(* IEC 61131-3 sources: test/SharedPlc, 5 files *)

(* ---- LPHD_Time.gvl ---- *)
VAR_GLOBAL
	DtTmAct 			: DT; 		(* --- Actual local time without summer time shift *)
	DtTmActSec 			: DINT;		(* --- Actual local time in second since 1.1.1970 *)
	DtTmActUtc 			: DT; 		(* --- Actual UTC Date and Time from the control system *)
	DtTmActUtcSec 		: DINT; 	(* --- Actual UTC Date and Time from the control system in seconds since 1.1.1970 *)
	DtTmShStri			: STRING;	(* --- Timezone shift from UTC in the format 'GMT+00:00'*)
	DtTmShSec			: DINT;		(* --- Timezone shift in seconds *)
	DtTmShM				: DINT;		(* --- Timezone shift in minutes *)
END_VAR

(* ---- SwitchIO.st ---- *)
FUNCTION SwitchIO : BOOL
VAR_INPUT
                Val:        BOOL;
                Switch: DINT;
END_VAR

VAR

END_VAR

CASE Switch OF
                -1: SwitchIO := Val XOR TRUE;
                0:  SwitchIO := FALSE;
                1:  SwitchIO := TRUE;
                2:  SwitchIO := Val;
END_CASE

END_FUNCTION

(* ---- TonSec.st ---- *)
FUNCTION_BLOCK TonSec
VAR_INPUT
	In		: BOOL;
	PTs		: DWORD; (* --- Time in seconds *)
END_VAR
VAR_OUTPUT
	ETs	:	DWORD;
	Q		: BOOL;
	PTDT	: DT;
	ETDT	: DT;	(* --- Time in seconds *)
END_VAR
VAR
	Str		: R_TRIG;
	StrTm 	: DT;
END_VAR

Str(S1 := In);
IF Str.Q0 THEN
	StrTm := DtTmActUtc;
END_IF

PTDT := UDINT_TO_DT(DT_TO_UDINT(StrTm) + PTs);
IF In THEN
	IF ETDT < PTDT   THEN

		ETDT := DtTmActUtc;
		ETs := PTs - (DT_TO_UDINT(PTDT) - DT_TO_UDINT(ETDT));
	END_IF

	IF ETDT >= PTDT THEN
		Q := TRUE;
	END_IF
ELSE
	ETs		:=	0;
	ETDT	:=	BYTE_TO_DT(0);
	Q		:=	FALSE;
END_IF

END_FUNCTION_BLOCK

(* ---- UpDnCnt.st ---- *)
FUNCTION_BLOCK UpDnCnt

VAR_INPUT
	IN		: BOOL;
	Cyc		: UDINT;
	RsCond	: INT;
END_VAR
VAR_OUTPUT
	OUT		: BOOL;
	CntEnd	: BOOL;
END_VAR
VAR
	Cnt: UDINT;
END_VAR

(* --- Reset Condition 0: Out will be FALSE, if IN FALSE *)
(* --- Reset Condition 1: Out will be FALSE, if IN FALSE and the time was counted down *)

IF (IN) THEN
	IF (Cnt >= Cyc) THEN
		Cnt := Cyc;
		OUT := TRUE;
	ELSE
		Cnt := Cnt + 1;
	END_IF
ELSE
	IF (Cnt <= 0) THEN
		Cnt := 0;
		OUT := FALSE;
	ELSE
		Cnt := Cnt - 1;
	END_IF

	IF(RsCond = 0)THEN
		OUT := FALSE;
	END_IF
END_IF

CntEnd := Cnt >= Cyc;

END_FUNCTION_BLOCK

(* ---- TimeHdl.st ---- *)
PROGRAM TimeHdl
VAR
	timespec_microseconds_Ds	: timespec_microseconds;
	DtOld						: DT;
	DtTmActLoc					: DT;
	SysTmUsec					: UDINT;
	USecOld						: UDINT;
	USecAct						:UDINT;
END_VAR
VAR_OUTPUT
	DTMS : DTMS;
END_VAR

(* --- Get time from system *)
clock_gettime(ADR(timespec_microseconds_Ds),TIMESPEC_RESOLUTION_MICROSECONDS,CLOCK_ID_CLOCK_RTCNANO);

DtTmActLoc := timespec_microseconds_Ds.dateAndTime;

(* WppTimeShiftMinutes_GDi: Wird aus der Monitoring Vorgabe in TimeZone_GpSt geholt *)
DTMS.DateAndTime := DINT_TO_DT(DT_TO_DINT(DtTmActLoc) + DtTmShSec);

(* --- SysTmUsec are in s from CPU start *)
SysTmUsec			:= timespec_microseconds_Ds.microseconds;
USecAct  			:= ((USecAct + ABS(SysTmUsec - USecOld)) MOD 1000000);
DTMS.Millisecond 	:= UDINT_TO_UINT(USecAct / 1000);

IF (TIME_TO_BOOL (ABS(DTMS.DateAndTime - DtOld))) THEN
	USecAct := 0;
END_IF

USecOld := SysTmUsec;
DtOld := DTMS.DateAndTime;

DtTmAct 		:= DTMS.DateAndTime;				(* --- Actual local time without summer time shift *)
DtTmActSec 		:= DT_TO_UDINT(DtTmAct);			(* --- Actual local time in second since 1.1.1970 *)
DtTmActUtc 		:= Tcs_RTC_GetDateAndTime(0);		(* --- Actual UTC Date and Time from the control system *)
DtTmActUtcSec 	:= DT_TO_UDINT(DtTmActUtc);			(* --- Actual UTC Date and Time from the control system in seconds since 1.1.1970 *)

(* TODO: check where we can get this information*)
(*ActDateAndTimeDST_GDt 	:=*) 						(* --- Actual local time with summer time shift *)

(* TODO: This information must be read out of the system/parameter - for start fix to GMT+00:00*)
DtTmShStri := 'GMT+00:00';	(* --- Time shift from UTC in the format 'GMT+00:00'*)
(*DtTmShM :=*) (*TODO: Calculate time shift from UTC in minutes *)

(*IecTmUtc := ;*)	(* TODO: Get IEC norm timestamp *)

END_PROGRAM
